# B&R Automation Studio project TD52 (part 23)

### module_AGPara.typ
```iecst
TYPE
	PARA_AG_struct : 	STRUCT
		tiFreshOilPump_Delay : TIME := T#5s; (*PARA [15065]  OilFill V4.14*) (*OldName: NewPV V4.14*)
		iOilRefill_Type : INT; (*PARA [xxxxx]  OilFill V4.14 prepared*) (*OldName: NewPV V4.14*)
		tiPostLub_Continuous : TIME; (*PARA [14930]  Turbocharger post lubrication - Duration of the continuous phase [s]*) (*OldName: new PV; Cycle:5*) (*V04.12.00.00*)
		iNum_PostLub_Interval : INT; (*PARA [14931]  Turbocharger post lubrication - number of intervals*) (*OldName: new PV; Cycle:5*) (*V04.12.00.00*)
		tiPostLub_PumpOff : TIME; (*PARA [14932]  Turbocharger post lubrication - Duration oil pump OFF [s]*) (*OldName: new PV; Cycle:5*) (*V04.12.00.00*)
		tiPostLub_PumpOn : TIME; (*PARA [14933]  Turbocharger post lubrication - Duration oil pump ON [s]*) (*OldName: new PV; Cycle:5*) (*V04.12.00.00*)
		bOilTankMonitoring : BOOL; (*PARA [14893]  OilTank V4.12*) (*OldName: NewPV V4.12*)
		rFreshOilTank_Type : REAL; (*PARA [14867]  OilTank V4.12*) (*OldName: NewPV V4.12*)
		rFreshOilTank_Length : REAL; (*PARA [14868]  OilTank V4.12*) (*OldName: NewPV V4.12*)
		rFreshOilTank_Height : REAL; (*PARA [14869]  OilTank V4.12*) (*OldName: NewPV V4.12*)
		rFreshOilTank_Witdh : REAL; (*PARA [14870]  OilTank V4.12*) (*OldName: NewPV V4.12*)
		rFreshOilTank_SensorPos : REAL; (*PARA [14871]  OilTank V4.12*) (*OldName: NewPV V4.12*)
		rWasteOilTank_Type : REAL; (*PARA [14876]  OilTank V4.12*) (*OldName: NewPV V4.12*)
		rWasteOilTank_Length : REAL; (*PARA [14877]  OilTank V4.12*) (*OldName: NewPV V4.12*)
		rWasteOilTank_Height : REAL; (*PARA [14878]  OilTank V4.12*) (*OldName: NewPV V4.12*)
		rWasteOilTank_Witdh : REAL; (*PARA [14879]  OilTank V4.12*) (*OldName: NewPV V4.12*)
		rWasteOilTank_SensorPos : REAL; (*PARA [14880]  OilTank V4.12*) (*OldName: NewPV V4.12*)
		rFreshOilTank_VolumeTotal : REAL; (*PARA [14894]  OilTank V4.12*) (*OldName: NewPV V4.12*)
		rWasteOilTank_VolumeTotal : REAL; (*PARA [14898]  OilTank V4.12*) (*OldName: NewPV V4.12*)
		rDayOilTank_VolumeTotal : REAL; (*PARA [14899]  OilTank V4.12*) (*OldName: NewPV V4.12*)
		rDayOilTank_Type : REAL; (*PARA [14885]  OilTank V4.12*) (*OldName: NewPV V4.12*)
		rDayOilTank_Length : REAL; (*PARA [14886]  OilTank V4.12*) (*OldName: NewPV V4.12*)
		rDayOilTank_Height : REAL; (*PARA [14887]  OilTank V4.12*) (*OldName: NewPV V4.12*)
		rDayOilTank_Witdh : REAL; (*PARA [14888]  OilTank V4.12*) (*OldName: NewPV V4.12*)
		rDayOilTank_SensorPos : REAL; (*PARA [14889]  OilTank V4.12*) (*OldName: NewPV V4.12*)
		rV_FreshOilTank_LimHi : REAL; (*PARA [14875]  OilTank V4.12*) (*OldName: NewPV V4.12*)
		rV_FreshOilTank_LimLo : REAL; (*PARA [14874]  OilTank V4.12*) (*OldName: NewPV V4.12*)
		rV_DayOilTank_LimHi : REAL; (*PARA [14875]  OilTank V4.12*) (*OldName: NewPV V4.12*)
		rV_DayOilTank_LimLo : REAL; (*PARA [14874]  OilTank V4.12*) (*OldName: NewPV V4.12*)
		rV_WasteOilTank_LimHi : REAL; (*PARA [14883]  OilTank V4.12*) (*OldName: NewPV V4.12*)
		rFreshOilTank_ScalMin : REAL; (*PARA [14872] [HalIO takeover]  OilTank V24*) (*OldName: NewPV V4.12*)
		rFreshOilTank_ScalMax : REAL; (*PARA [14873] [HalIO takeover]  OilTank V24*) (*OldName: NewPV V4.12*)
		rWasteOilTank_ScalMin : REAL; (*PARA [14881] [HalIO takeover]  OilTank V24*) (*OldName: NewPV V4.12*)
		rWasteOilTank_ScalMax : REAL; (*PARA [14882] [HalIO takeover]  OilTank V24*) (*OldName: NewPV V4.12*)
		rDayOilTank_ScalMin : REAL; (*PARA [14890] [HalIO takeover]  OilTank V24*) (*OldName: NewPV V4.12*)
		rDayOilTank_ScalMax : REAL; (*PARA [14891] [HalIO takeover]  OilTank V24*) (*OldName: NewPV V4.12*)
		bER_VentColdCountryMode : BOOL; (*PARA [12246]: engine room ventilation cold country mode *) (*OldName:MRL_KL; Cycle:5*)
		bPurgecycle_Active : BOOL; (*PARA [12256]: purge cycle enable*) (*OldName:bPurgecycle; Cycle:5*)
		bVISA : BOOL; (*PARA [12259]: monitoring according VISA*) (*OldName:VISA; Cycle:5*)
		bTSTC_Exist : BOOL; (*PARA [10018]: Engine with TSTC *) (*OldName:b2StageTC; Cycle:5*)
		bEngTyp3_Prelub_Active : BOOL; (*PARA [10009]: prelubrication for engine typ 3 active *) (*OldName:BR3_VS_aktiv; Cycle:5*)
		bTC_PostLub_Active : BOOL; (*PARA [10015]: turbo charger post lubrication active *) (*OldName:new; Cycle:5*)
		bBS_Acc_Active : BOOL; (*PARA [12178]: accelerated black start active *) (*OldName:sel_black_start_15s; Cycle:5*)
		bSel_TwoN2Valves : BOOL; (*PARA [11313]: select exhaust gas scavenging with 2 nitrogen*) (* OldName:TwoN2Valves; Cycle:5*)
		bECWP_MechDriven : BOOL; (*PARA [10007]: engine cooling water pump mechanical driven*) (*OldName:sel_BR3_eMKWP; Cycle:5*)
		bTC_watercooled : BOOL; (*PARA [10016]: water cooled turbo charger *) (*OldName:ATL_H2O; Cycle:5*)
		iEng_Motortype : INT; (* Motor type of the engine *) (*OldName:iMotortyp; Cycle:5*)
		rN_ECWP_Set : REAL; (*PARA [10032]: speed engine cooling water pump setpoint *) (* OldName:GW_SP_MKWP; Cycle:5*)
		rN_EngStart_HyHi : REAL; (*PARA [11295]: speed engine start limit high hysteresis *) (*OldName:HY_DREHZ; Cycle:5*)
		rN_EngStart_HyHiHi : REAL; (*PARA [11507]: speed engine start limit high high hysteresis *) (*OldName:HY_HDREHZ; Cycle:5*)
		rN_EngStartMon_LimHi : REAL; (*PARA [12068]: speed engine start monitoring limit high*) (*OldName:GW_STRDRE; Cycle:5*) (*V04.13.00.00*)
		rN_EngStart_LimHi : REAL; (*PARA [11296]: speed engine start limit high *) (*OldName:GW_DREHZ; Cycle:5*)
		rN_EngStart_LimHiHi : REAL; (*PARA [11508]: speed engine start limit high high *) (*OldName:GW_HDREHZ; Cycle:5*)
		rPr_CC_LimHiHi : REAL; (*PARA [10060]: pressure crank case limit high high *) (*OldName:GW_p_CC_high; Cycle:5*)
		bPr_CC_MS_Exist : BOOL; (*PARA [10013]: pressure crank case measuring signal exist *) (*OldName:p_CC_a; Cycle:5*)
		rPr_Prel1EOP_LimHi : REAL; (*PARA [10076]: prelubrication pressure limit for 1 pump*) (*OldName:GW_VSD1; Cycle:5*)
		rPr_Prel1EOP_HyHi : REAL; (*PARA [10075]: prelubrication pressure limit for 1 pump hysteresis*) (*OldName:HY_VSD1; Cycle:5*)
		rPr_Prel2EOP_LimHi : REAL; (*PARA [10078]: prelubrication pressure limit for 2 pump*) (*OldName:GW_VSD2; Cycle:5*)
		rPr_Prel2EOP_HyHi : REAL; (*PARA [10077]: prelubrication pressure limit for 2 pump hysteresis*) (*OldName:HY_VSD2; Cycle:5*)
		rPr_TCOF_PrelubMin : REAL; (*PARA [10087]: TC - filter outlet prelubrication pressure minimum*) (*OldName:GW_ODTC_MI_PREL; Cycle:5*)
		rPr_TCOF_PrelubHyMin : REAL; (*PARA [10086]: filter outlet prelubrication pressure minimum hysteresis*) (*OldName:HY_ODTC_MI_PREL; Cycle:5*)
		rT_ECW_PreH_HyOFF : REAL; (*PARA [10088]: temperature engine cooling water preheating limit off hysteresis *) (*OldName:HY_VORW; Cycle:5*)
		rT_ECW_PreH_LimOFF : REAL; (*PARA [10089]: temperature engine cooling water preheating limit off *) (*OldName:GW_VORW; Cycle:5*)
		bCtr_CC : BOOL; (*PARA [12644]: visibility crank case pressure controller*) (*OldName:new; Cycle:5*)
		bCtr_ECW : BOOL; (*PARA [10005]: visibility engine cooling water controller*) (*OldName:new; Cycle:5*)
		tCtr_CC : _tGeACtrPara; (*Para controller actual speed*) (*OldName:new; Cycle:5*)
		tCtr_ECW : _tGeACtrPara; (*Para controller engine cooling water temperature*) (*OldName:new; Cycle:5*)
		bTCOP_Visible : BOOL; (*PARA [10017]: turbo charger oil pump visible*) (*OldName:bVisuTCPump; Cycle:5*)
		bEOP_AC_Visible : BOOL; (*PARA [10010]: engine oil pump prelube AC visible*) (*OldName:bVisuACPump; Cycle:5*)
		bEOP_DC_Visible : BOOL; (*PARA [10011]: engine oil pump DC visible*) (*OldName:bVisuDCPump; Cycle:5*)
		bECW_PreH_Visible : BOOL; (*PARA [10006]: engine cooling water preheating visible*) (*OldName:bPreHeat; Cycle:5*)
		bECWP_PreH_Visible : BOOL; (*PARA [10008]: engine cooling water preheating pump visible*) (*OldName:bPreHeatWatPump; Cycle:5*)
		b_EOF_DiffMonActive : BOOL; (*PARA [10002]: Oil pressure before oil filter active M.03-PI-002(NUP29)*) (*OldName:bOilFilterPressAct; Cycle:5*)
		rN_EOP_Lim1 : REAL; (*PARA [10033]: Engine Speed 1 for oil pressure monitoring*) (*OldName:DR_ODR_1; Cycle:5*)
		rPr_EOP_HyMin : REAL; (*PARA [10070]: Oil pressure mimimum hysteresis*) (*OldName:HY_ODRA; Cycle:5*)
		rPr_EOP_HyLim1 : REAL; (*PARA [10068]: Oil pressure limit 1 hysteresis*) (*OldName:HY_ODGW1; Cycle:5*)
		rPr_EOP_LimMax : REAL; (*PARA [10072]: Oil pressure maximum*) (*OldName:GW_ODR_MAX; Cycle:5*)
		rPr_EOP_HyMax : REAL; (*PARA [10069]: Oil pressure maximum hysteresis*) (*OldName:HY_ODR_MAX; Cycle:5*)
		rPr_EOP_LimSpeed2 : REAL; (*PARA [10074]: Limit oil pressure at engine speed 2*) (*OldName:GW_ODR_2; Cycle:5*)
		rN_EngNom : REAL; (*PARA [12128]: engine nominal speed*) (*OldName:n_nenn; Cycle:5*)
		rN_TCOF_Lim1 : REAL; (*PARA [10037]: TC - filter outlet pressure minimum speed scale value 1 for pressure monitoring*) (*OldName:DR_ODR_TC_1; Cycle:5*)
		rN_TCOF_Lim2 : REAL; (*PARA [10038]: TC - filter outlet pressure minimum speed scale value 2 for pressure monitoring*) (*OldName:DR_ODR_TC_2; Cycle:5*)
		rPr_TCOF_LimSpeed1 : REAL; (*PARA [10082]: TC - filter outlet pressure minimum oil limit value 1 for pressure monitoring*) (*OldName:GW_ODR_TC_1; Cycle:5*)
		rPr_TCOF_LimSpeed2 : REAL; (*PARA [10083]: TC - filter outlet pressure minimum oil limit value 2 for pressure monitoring*) (*OldName:GW_ODR_TC_2; Cycle:5*)
		rPr_TCOF_HyMin : REAL; (*PARA [10080]: TC - filter outlet pressure minimum hysteresis*) (*OldName:HY_ODTC_MI; Cycle:5*)
		rPr_TCOF_MinWarn : REAL; (*PARA [10085]: TC - filter outlet pressure minimum warning*) (*OldName:GW_ODTC_MI_W; Cycle:5*)
		rPr_TCOF_HyMinWarn : REAL; (*PARA [10081]: TC - filter outlet pressure minimum warning hysteresis*) (*OldName:HY_ODTC_MI_W; Cycle:5*)
		rPr_TCOF_Max : REAL; (*PARA [10084]: TC - filter outlet pressure maximum*) (*OldName:GW_ODTC_MA; Cycle:5*)
		rPr_TCOF_HyMax : REAL; (*PARA [10079]: TC - filter outlet pressure maximum hysteresis*) (*OldName:HY_ODTC_MA; Cycle:5*)
		rT_EO_PreheatMin : REAL; (*PARA [10093]: Limit start oil pre warning*) (*OldName:GW_OILVORW; Cycle:5*)
		rT_EO_PreheatHyMin : REAL; (*PARA [10092]: Limit start oil pre warning hysteresis*) (*OldName:HY_OILVORW; Cycle:5*)
		rT_EO_LimMin : REAL; (*PARA [10091]: Oil temperature minimum *) (*OldName:GW_OTMI; Cycle:5*)
		rT_EO_LimHyMin : REAL; (*PARA [10090]: Oil temperature minimum hysteresis*) (*OldName:HY_OTMI; Cycle:5*)
		b_TCEO_HE2Ena : BOOL; (*PARA [10004]: Activate picture for second oil heat exchanger*) (*OldName:bVisuOil2stage; Cycle:5*)
		rEOP_PreLube_Set : REAL; (*PARA [12673]: speed setpoint engine oil pump prelubrication (frequency converter)*) (*OldName:GW_SP_OILP_PREL; Cycle:5*)
		rEOP_PreHeat_Set : REAL; (*PARA [12674]: speed setpoint engine oil pump preheating (frequency converter)*) (*OldName:GW_SP_OILP_PREH; Cycle:5*)
		r_OV_LimOpen : REAL; (*PARA [10029]: Limit oil valve open*) (*OldName:GW_OELVA; Cycle:5*)
		r_OV_HyLimOpen : REAL; (*PARA [10027]: Limit oil valve open hysteresis*) (*OldName:HY_OELVA; Cycle:5*)
		r_OV_LimClose : REAL; (*PARA [10028]: Limit oil valve close*) (*OldName:GW_OELVZ; Cycle:5*)
		r_OV_HyLimClose : REAL; (*PARA [10026]: Limit oil valve close hysteresis*) (*OldName:HY_OELVZ; Cycle:5*)
		r_EO_LevelLimMax : REAL; (*PARA [10024]: Oil level maximum*) (*OldName:GW_OMAX; Cycle:5*)
		r_EO_W_LevelLimMax : REAL; (*PARA [14966]: Oil level maximum warning [%]*) (*OldName: newPV ; Cycle:5*) (*V04.13.00.00*)
		r_EO_W_LevelLimMin : REAL; (*PARA [13964]: Oil level minimum warning*) (*OldName: newPV ; Cycle:5*)
		r_EO_LevelHyLimMax : REAL; (*PARA [10022]: Oil level maximum hysteresis*) (*OldName:HY_OMAX; Cycle:5*)
		r_EO_LevelLimMin : REAL; (*PARA [10025]: Oil level minimum*) (*OldName:GW_OMIN; Cycle:5*)
		r_EO_LevelHyLimMin : REAL; (*PARA [10023]: Oil level minimum hysteresis*) (*OldName:HY_OMIN; Cycle:5*)
		rT_EOF_DiffMonRel : REAL; (*PARA [10094]: Oil filter differential pressure monitoring - Oil temperature for release [degC]*) (*OldName:ssOilFilterPOilTemp; Cycle:5*)
		rPr_EOP_LimSpeed1 : REAL; (*PARA [10073]: Limit oil pressure at engine speed 1*) (*OldName:GW_ODR_1; Cycle:5*)
		rPr_EOP_Lim1 : REAL; (*PARA [10071]: Oil pressure limit 1*) (*OldName:GW_ODGW1; Cycle:5*)
		rPr_LimHeatRel : REAL; (*PARA [12807]: Pressure limit for release heating*) (*OldName:GW_druck_heizfreigabe; Cycle:5*)
		rN_EOP_Lim2 : REAL; (*PARA [10034]: Engine Speed 2 for oil pressure monitoring*) (*OldName:DR_ODR_2; Cycle:5*)
		b_OilActive : BOOL; (*PARA [10003]: oil counter exist*) (*OldName:bExistOilCounter; Cycle:5*)
		iNum_OilPulse : INT; (*PARA [10020]: Impulse valency*) (*OldName:ssOilPulseValue; Cycle:5*)
		bCtr_EOVal_Active : BOOL; (*PARA [12615]: engine oil cooler valve controller Active*) (*OldName:new; Cycle:5*)
		rT_EOP_LimMax : REAL; (*PARA [10097]: Oil temperature maximum *) (*OldName:GW_OTMA; Cycle:5*)
		rT_EOP_HyMax : REAL; (*PARA [10095]: Oil temperature maximum hysteresis*) (*OldName:HY_OTMA; Cycle:5*)
		rT_EOP_HyRelLoad : REAL; (*PARA [10096]: Oil temperature release load, load enabling hysteresis*) (*OldName:HY_OT_LFG; Cycle:5*)
		rT_EOP_LimRelLoad : REAL; (*PARA [10098]: oil temperature release load*) (*OldName:GW_OT_LFG; Cycle:5*)
		tCtr_EOVal : _tGeACtrPara; (*Para: structure for engine oil controller*) (*OldName:new; Cycle:5*)
		rP_Red_T_Oil_Start : REAL; (*PARA [10049]: power reduction oil temp. start [°C]*) (*OldName:Pred_OT_start; Cycle:5*)
		rP_Red_T_Oil_Rate : REAL; (*PARA [10048]: power reduction oil temp.rate [%]*) (*OldName:Pred_OT_rate; Cycle:5*)
		rPr_EOF_DiffMonLimit1 : REAL; (*PARA [10065]: Oil filter differential pressure monitoring - Oil filter service life limit [bar]*) (*OldName:ssOilFilterLimit1; Cycle:5*)
		rPr_EOF_DiffMonLimit2 : REAL; (*PARA [10066]: Oil filter differential pressure monitoring - Oil filter to be replaced [bar]*) (*OldName:ssOilFilterLimit2; Cycle:5*)
		rPr_EOF_DiffMonLimit3 : REAL; (*PARA [10067]: Oil filter differential pressure monitoring - Shutdown [bar]*) (*OldName:ssOilFilterLimit3; Cycle:5*)
		i_OilRefillBlocked : DINT; (*PARA [10019]: Number of operating hours until next refill*) (*OldName:slBlockOilRefill_Bh; Cycle:5*)
		bEO_Level_Active : BOOL; (*PARA [12805]: Engine oil level measuring active*) (*OldName:ALM[2576].ENABLE; Cycle:5*)
		bPr_EOF_After_Active : BOOL; (*PARA [12722]: Oil pressure after oil filter active M.03-PI-057*) (*OldName:new PV; Cycle:5*)
		bGridCode_Active : BOOL; (*PARA [11055]: Gride Code active*) (*OldName:bGridCode; Cycle:5*)
		bPr_TCOaF_Active : BOOL; (*PARA [10014]: pressure oil turbo charger after filter signal active*) (*OldName:new; Cycle:5*)
		bCtr_EOVal_LT_Active : BOOL; (*PARA [12705]: engine oil cooler LT valve controller Active*) (*OldName:new; Cycle:5*)
		tCtr_EOVal_LT : _tGeACtrPara; (*Para: structure for engine oil controller*)
		bT_EOaPump_Active : BOOL; (*PARA [12723]: engine oil temperature after pump active*)
		bPr_Oil_LPTC_In_A : BOOL; (*PARA [12724]: oil pressure LP turbo charger A inlet measuring active*)
		bPr_Oil_LPTC_In_B : BOOL; (*PARA [12725]: oil pressure LP turbo charger B inlet measuring active*)
		bPr_f_BbFilt_Exist : BOOL; (*PARA [12566]: Druck vor Blow-by Filter aktiv, Pressure before Blow-by filter	*)
		rP_CC_MonActive_LimHi : REAL; (*PARA [10047]: -Visu only- Kurbelgehaeusedruckueberwachung aktiv, Crank Case Pressure check active [% Pnom]*) (*Oldname: GW_P_CCM, Cycle:5 *)
		rPr_CC_Lo : REAL; (*PARA [12560]: Kurbelgehaeusedruck Minimum - Warnung, Crank Case Pressure Minimum Warning [bar]*)
		rPr_CC_Hi : REAL; (*PARA [12561]: Crank case pressure high - warning [bar]*)
		rP_Red_CC : REAL; (*PARA [12564]: Power reduction by Crank case pressure [% Pnom]*)
		rPc_BbBlower_Hi : REAL; (*PARA [12565]: Operating point blow by blower maximum [%]*)
		bPr_a_BbFilt_Exist : BOOL; (*PARA [12571]: pressure after blow by filter exist*)
		rDPr_BbFilt_Pstart : REAL; (*PARA [12618]: Blow by filter difference pressure start point for monitoring [% Pnom]*)
		rDPr_BbFilt_Lo_P1 : REAL; (*PARA [12619]: Blow by filter difference pressure new filter - lower load point [bar]*)
		rDPr_BbFilt_Lo_P2 : REAL; (*PARA [12620]: Blow by filter difference pressure new filter - full load [bar]*)
		rDPr_BbFilt_Hi_P1 : REAL; (*PARA [12621]: Blow by filter difference pressure charged filter - lower load point [bar]*)
		rDPr_BbFilt_Hi_P2 : REAL; (*PARA [12622]: Blow by filter difference pressure charged filter - full load [bar]*)
		tiPr_CC_Hi : TIME; (*PARA [12562]: Crank case pressure high - time until warning [s]*)
		tiPr_CC_HiHi : TIME; (*PARA [12563]: Crank case pressure high - time until error [s]*)
		bT_EO_Pan_Active : BOOL; (*PARA [12747]: engine oil temperature oil pan active*)
		bPr_TCObF_Active : BOOL; (*PARA [12742]: turbocharger oil pressure before filter active*)
		bPr_AirStarter_Tank_Exist : BOOL; (*PARA [12648]: air starter tank pressure exist *)
		rPr_AirStarter_Tank_Lo : REAL; (*PARA [10055]: air starter tank pressure minimum [bar] *)
		bPr_AirStarter_Supply_Exist : BOOL; (*PARA [12651]: air starter supply pressure exist	*)
		rPr_AirStarter_Supply_LoLo : REAL; (*PARA [10053]: air starter supply pressure minimum - error [bar] *)
		rPr_AirStarter_Supply_HiHi : REAL; (*PARA [10052]: air starter supply pressure maximum - error [bar] *)
		bN_AirStarter_Exist : BOOL; (*PARA [12654]: air starter speed exist	*)
		tiAirStarter_OnTime : TIME; (*PARA [10119]: air starter ON Time / Engaging Time (Einspurzeit) [ms]*)
		tiTC_Postlub : TIME; (*PARA [12775]: turbo charger postlube duration for water cooled TC [ms]*)
		bManAuxCtr_Active : BOOL; (*PARA [12917]: Manual operating auxiliaries control is active*)
		tiManAuxCtr_Max : TIME; (*PARA [12916]: Maximum release time of manual operating auxiliaries control*)
		tiFreshOilPump_Intervall : TIME; (*PARA [xxxxx]: time for run time intervall fresh oil pump*) (*OldName: NewPV V4.14*)
		tiFreshOilPump_Pause : TIME; (*PARA [xxxxx]: time for stop intervall fresh oil pump*) (*OldName: NewPV V4.14  SEE ALSO -->PARA [13308]: time for run time overload fresh oil pump*)
		tiFreshOilPump_RTC_Time : TIME; (*PARA [13308]: time for run time overload fresh oil pump*)
		rP_Red_TransformerWarning_Rate : REAL; (*PARA [13270]: transformer power reduction setpoint*)
		bP_Red_TransformerWarning_Sel : BOOL; (*PARA [13269]: activation transformer power reduction*)
		bPr_f_BbFilt_A_Exist : BOOL; (*PARA [13265]: pressure before blow-by filter aktiv*)
		bPr_f_BbFilt_B_Exist : BOOL; (*PARA [13266]: pressure before blow-by filter aktiv*)
		bPr_a_BbFilt_A_Exist : BOOL; (*PARA [13267]: pressure after blow by filter exist*)
		bPr_a_BbFilt_B_Exist : BOOL; (*PARA [13268]: pressure after blow by filter exist*)
		bCDP_Active : BOOL; (*PARA [13182]: Kondensorpumpe active*)
		bPr_EOaP_Active : BOOL; (*PARA [13398]: engine oil pressure after pump active M.03-PI-007*)
		rPr_EOaP_LimHi : REAL; (*PARA [13399]: engine oil pressure after pump limit high M.03-PI-007*)
		rPr_EOaP_LimHiHi : REAL; (*PARA [13400]: engine oil pressure after pump limit high high M.03-PI-007*)
		bOilFiltUnit_Exist : BOOL; (*PARA [13470]: oil filter unit existing*)
		bPr_OFUbFilt_Active : BOOL; (*PARA [13471]: pressure oil filter unit before filter M.03-PI-011*)
		bPr_OFUaFilt_Active : BOOL; (*PARA [13474]: pressure oil filter unit after filter M.03-PI-012*)
		bServicePrelub : BOOL; (*PARA [13827]: prelube with both oil pumps - service button*)
		rPr_EObF_LimHi : REAL; (*PARA [13962]: Oil pressure filter inlet maximum warning [bar] M.03-PI-002(NUP29)*)
		rPr_EObF_LimHiHi : REAL; (*PARA [13963]: Oil pressure filter inlet maximum alarm [bar] M.03-PI-002(NUP29)*)
		bPr_OFUbCentrifuge_Active : BOOL; (*PARA [13631]: pressure oil filter unit before centrifuge M.03-PI-008*)
		rDPr_OFU_Filt_LimHi : REAL; (*PARA [13477]: difference pressure oil filter unit - limit high*)
		rPr_OFUbFilt_Hi : REAL; (*PARA [13630]: pressure oil filter unit before filter - limit high*)
		rPr_OFUbCentrifuge_Hi : REAL; (*PARA [13634]: pressure oil filter unit before centrifuge - limit high*)
		bPr_TCO_Active : BOOL; (*PARA [14114]: pressure oil before turbo charger [bar]*)
		tiFSPreL : TIME; (*PARA [14166]: permanent prelubrication minimum operating time for faststart release*)
		rPr_TCO_FSPreL_LimHi : REAL; (*PARA [14167]: pressure oil before turbo charger limit high - permanent prelubrication [bar]*)
		rPr_TCO_FSPreL_LimLo : REAL; (*PARA [14169]: pressure oil before turbo charger limit low - fast start [bar]*)
		rN_TCO_FS : REAL; (*PARA [14168]: speed point fast start [rpm]*)
		rT_EO_PreH_FS_Min : REAL; (*PARA [14170]: limit low start oil preheating warning/fast start [°C]*)
		rT_EO_PreH_FS_HyMin : REAL; (*PARA [14171]: Limit low start oil preheating warning hysteresis/fast start [°C]*)
		rPr_EO_PreH_LimLo : REAL; (*Para: engine oil pressure limit low preheating [bar]*)
		rPr_EO_FSPreL_LimLo : REAL; (*PARA [14165]: engine oil pressure limit low permanent prelubrication [bar]*)
		tiReEngage : TIME; (*PARA [14065]: delay reengagement air starter*)
		bFSPreL_Act : BOOL; (*PARA [14208]: permanent prelubrication active*)
		bBbOp_EOP : BOOL; (*PARA [14172]: blowby fan operation with engine oil pump*)
		bPreLub_Interval_Enable : BOOL; (*PARA [14066]: Interval pre lubrication enable *)
		tiPreLub_Interval : TIME; (*PARA [13965]: interval time pre lubrication *)
		rPr_PreLub_Interval_Lim : REAL; (*PARA [13966]: engine interval pre lubrication pressure limit *)
		rU_StarterBat_Lo : REAL; (*PARA [13989]: Starter battery voltage minimum (UL) while battery test*)
		rU_StarterBat_Hi : REAL; (*PARA [13990]: Starter battery voltage high*)
		bACP_Enable : BOOL; (*PARA [13984]: Enable Active Cooling *)
		rT_ACP_ECW_sp : REAL; (*PARA [13985]: Active cooling program setpoint temperature engine cooling water system *)
		rT_ACP_EO_sp : REAL; (*PARA [13986]: Active cooling program setpoint temperature engine cooling water system *)
		rT_ACP_AirER_sp : REAL; (*PARA [13987]: Active cooling program setpoint temperature engine room ventilation *)
		rT_EO_LimHiHi : REAL; (*PARA [14180]: Oil temperature high high//SWAT920/5*)
		bECW_PreH_Fast : BOOL; (*PARA [14349]: Fast ECW heat-up active*)
		rT_ECW_HydrPreH_LimLo : REAL; (*PARA [14350]: Delta hydraulic pre-heating warning [°C]*)
		iECW_PreH_Int_Visible : INT; (*PARA [11902]: Pre-heating type jacket water (formerly: Internal heating)*)
		bT_HW_Su_PreH_ECW_Active : BOOL; (*PARA [12912]: Heating water temperature supply hydraulic ECW preheating measuring active*)
		bRedHWP_Active : BOOL; (*PARA [14345]: Activate redundant pump control for heating water pump *)
		bRedCCWP_Active : BOOL; (*PARA [14347]: Activate redundant pump control for charge cooler water pump *)
		bRedCC2WP_Active : BOOL; (*PARA [14346]: Activate redundant pump control for charge cooler 2 water pump *)
		bRedEmCWP_Active : BOOL; (*PARA [14348]: Activate redundant pump control for emergency cooler water pump *)
		iCnt_TC_Inspection_Hi : DINT; (*PARA [14408]: Threshold for turbocharger inspection after number of failed post cooling cycles*)
		rPr_TC_EOF_After_Avg_Lo : REAL; (*PARA [14409]: Lower threshold average oil pressure for TC post cooling*)
		rPr_TC_Oil_CoolDownInterrupt_Lo : REAL; (*PARA [14410]: Lower threshold oil pressure for OCTC post cooling interruption*)
		bDPr_ECWP_Mon_Active : BOOL; (*PARA [14425]: Measurement cooling water difference pressure over ECW pump active*)
		rDPr_ECWP_LoLo : REAL; (*PARA [14428]: Difference pressure cooling water over ECW pump minimum*)
		tiAirST_Interrupt : TIME; (*PARA [14445]: Air starter start up time for interrupting blocked start valve*)
		bBbBlower_Off_Active : BOOL; (*PARA [14483]: Blow-by blower reduced operation mode*)
		rP_Norm_BbBlower_off : REAL; (*PARA [14484]: Engine power limit for blow by blower off [% Pnom]*)
		tiPr_CC_HiWarn : TIME; (*PARA [14485]: Crankcase pressure maximum  delay until warning [s]*)
		tiPreLube : TIME; (*PARA [14504]: Prelubrication duration (normal prelube, not permanent)*)
		bEO_Management_Active : BOOL; (*PARA [14496]: oil management function active*)
		bCW_Management_Active : BOOL; (*PARA [14497]: coolant management function active*)
		iEO_PreH_Int_Visible : INT; (*PARA [14503]: Pre-heating type engine oil (formerly: Internal heating)*)
		iBatMon_Mode : INT; (*PARA [14490]: Battery voltage monitoring mode*)
		rU_BufferBat_Lo : REAL; (*PARA [14491]: Buffer battery voltage minimum (UL) while battery test*)
		rU_BufferBat_Idle_Lo : REAL; (*PARA [14492]: Buffer battery voltage minimum idle voltage (U0)*)
		rU_StarterBat_Idle_Lo : REAL; (*PARA [14493]: Starter battery voltage minimum idle voltage (U0)*)
		rU_StarterBat_Crank_Lo : REAL; (*PARA [14494]: Starter battery voltage minimum starter cranking (UL)*)
		tiU_StarterBat_MeasDelay : TIME; (*PARA [14501]: Test begin starter battery voltage starter cranking (UL)*)
		tiU_StarterBat_MeasTime : TIME; (*PARA [14502]: Test duration starter battery voltage starter cranking (UL)*)
		rPr_OFUbCentrifuge_Lo : REAL; (*PARA [14734]: Oil pressure oil centrifuge inlet minimum warning [bar]*)
		iOQS_Config : UINT; (*PARA [14726]: Oil quality sensor configuration*)
		rOQS_OC_ScalFreshOil : REAL; (*PARA [14727]: Oil quality sensor: Oil condition value fresh oil (=100% oil quality) [%]*)
		rOQS_OC_ScalAgedOil : REAL; (*PARA [14728]: Oil quality sensor: Oil condition value aged oil (=0% oil quality) [%]*)
		rOilQual_OQS_OC_LimLo : REAL; (*PARA [14729]: Oil quality sensor: Limit oil quality warning [%]*)
		rOilQual_OQS_OC_LimLo1 : REAL; (*PARA [14731]: Oil quality sensor: Limit oil quality critical warning [%]*)
		rOilQualTendency_OQS_OC_LimHi : REAL; (*PARA [14730]: Oil quality sensor: Limit oil quality tendency warning [%/100oph]*)
		rOilQualTendency_OQS_OC_LimHi1 : REAL; (*PARA [14732]: Oil quality sensor: Limit oil quality tendency critical warning [%/100oph]*)
		iOilSamplingNomOh : DINT; (*PARA [14733]: Oil quality sensor: Regular oil sampling interval [oph]*)
		rT_OQS_LimLo : REAL; (*PARA [14921]: Oil quality sensor: Limit oil quality operating temperature [degC]*)
		rU_StarterMonTtT_LimHi : REAL; (*PARA [14927]: Starter monitoring: Tooth to tooth upper limit starter battery voltage [V]*)
		rN_StarterMonTtT_LimLo : REAL; (*PARA [14928]: Starter monitoring: Tooth to tooth lower limit engine speed [rpm]*)
		tiStarterMonDuration : TIME; (*PARA [14929]: Starter monitoring: Tooth to tooth detection duration [s]*)
		bOilRefill_MonAct : BOOL; (*PARA [14967]: Oil refill - Monitoring active*) (*OldName: newPV ; Cycle:5*) (*V04.13.00.00*)
		rVol_OilRefill_Pct_EO_Level : REAL; (*PARA [14968]: Oil refill - Refill volume per % oil level [l]*) (*OldName: newPV ; Cycle:5*) (*V04.13.00.00*)
		rPc_OilRefill_VolTolerance : REAL; (*PARA [14969]: Oil refill - Refill volume tolerance [%]*) (*OldName: newPV ; Cycle:5*) (*V04.13.00.00*)
		rU_StarterMon_LimLo : REAL; (*PARA [15015]: Starter function voltage level [V]*) (*OldName: newPV ; Cycle:5*) (*V04.13.00.00*)
		tiStarterFunDuration : TIME; (*PARA [15016]: Starter function detection time [s]*) (*OldName: newPV ; Cycle:5*) (*V04.13.00.00*)
		bEO_PreH_Active : BOOL; (*PARA [15019]: Oil preheating active*) (*OldName: newPV ; Cycle:5*) (*V04.13.00.00*)
		rT_EO_PreH_EngStart : REAL; (*PARA [15020]: Oil preheating - Target temperature for engine start [degC]*) (*OldName: newPV ; Cycle:5*) (*V04.13.00.00*)
		rVolFlow_Marg : REAL; (*PARA [15071]: Volume flow margin [%]*) (*V04.14.00.00*)
		rVolEff_CrkSpeed : REAL; (*PARA [15073]: Volumetric efficiency at cranking speed [-]*) (*V04.14.00.00*)
		iVol_MinAir_SysPurge : UDINT; (*PARA [15074]: Minimum air volume required for system purge [lt]*) (*V04.14.00.00*)
		rST_Heatup_Fact : REAL; (*PARA [15075]: Starter heatup factor [s/s]*) (*V04.14.00.00*)
		tiST_CooldownConst : TIME; (*PARA [15076]: Starter cool down time constant [s]*) (*V04.14.00.00*)
		tiST_MaxDur_OverheatPrev : TIME; (*PARA [15077]: Maximum starting duration overheat prevention [s]*) (*V04.14.00.00*)
		rST_ReqOpTiAftCooldown : REAL; (*PARA [15078]: Required starter operating time after cooldown [%]*) (*V04.14.00.00*)
		iVol_PremxInSys : UDINT; (*PARA [15079]: Premixed volume of the engine intake system [lt]*) (*V04.14.00.00*)
		iVol_TolUnbrtMxMax : UDINT; (*PARA [15080]: Maximum tolerable unburnt mixture volume [lt]*) (*V04.14.00.00*)
		bEGScav_Active : BOOL; (*PARA [11303]: exhaust gas scavenging active *) (*OldName:sel_EGScav;Cycle:5*) (*V04.14.00.00*)
		tiEO_Refill_TimeMax : TIME; (*PARA [15067]: oil refill time maximum *) (*V04.14.00.00*)
		bEGScav_ifAuxV_ok : BOOL; (*PARA [11304]: exhaust gas scavenging if auxiliaries voltage supply ok*) (*OldName:sel_EGScav_if_AuxV_ok;Cycle:5*)
	END_STRUCT;
END_TYPE
```

### module_AGPerm.typ
```iecst
(********************************************************************
 * COPYRIGHT -- INNIO Company
 ********************************************************************
 * Paket: AuxiliariesGeneral
 * Datei: module_AGPerm.typ
 * Autor: zengeres
 * Erstellt: 14. Oktober 2013
 ********************************************************************
 * Datentypen des Pakets AuxiliariesGeneral
 ********************************************************************)

TYPE
	tPerm_AG_typ : 	STRUCT
		tStartStat : ARRAY[0..200]OF tStartStat_typ;
		StatCnt : DINT;
		rAG_PermValue1 : REAL; (*spare permanent value - replace with new vars of same lenght, when needed*)
		rAG_PermValue2 : REAL; (*spare permanent value - replace with new vars of same lenght, when needed*)
		rAG_PermValue3 : REAL; (*spare permanent value - replace with new vars of same lenght, when needed*)
		rAG_PermValue4 : REAL; (*spare permanent value - replace with new vars of same lenght, when needed*)
		rAG_PermValue5 : REAL; (*spare permanent value - replace with new vars of same lenght, when needed*)
		rAG_PermValue6 : REAL; (*spare permanent value - replace with new vars of same lenght, when needed*)
		rAG_PermValue7 : REAL; (*spare permanent value - replace with new vars of same lenght, when needed*)
		rAG_PermValue8 : REAL; (*spare permanent value - replace with new vars of same lenght, when needed*)
		rAG_PermValue9 : REAL; (*spare permanent value - replace with new vars of same lenght, when needed*)
		rAG_PermValue10 : REAL; (*spare permanent value - replace with new vars of same lenght, when needed*)
	END_STRUCT;
	tStartStat_typ : 	STRUCT
		tiStartTime : RTCtime_typ;
		tiStarterON_Max : TIME;
		tiStarterOFF : TIME;
		tiStartScav : TIME;
		rN_EngStart : REAL;
		tiStartDuration : TIME;
		iStartID : DINT;
		bStartSuccess : BOOL;
	END_STRUCT;
END_TYPE
```

### module_AG.var
```iecst
VAR
	IN_AG : IN_AG_struct;
	OUT_AG : OUT_AG_struct;
	MM2VIS : MM2VIS_struct;
	VIS2MM : VIS2MM_struct;
	Para : PARA_AG_struct;
	ParaFactoryDefault : PARA_AG_struct;
	pm : PARA_AG_struct;
	tCtr_ECW_In : _tGeACtrIn; (*engine cooling water controller*)
	tCtr_ECW_Out : _tGeACtrOut; (*engine cooling water controller*)
	xCtr_ECW : GeACtr; (*engine cooling water controller*)
	xEngType : EngType;
	bEOVal_DemOpen : BOOL := FALSE; (*demand for oil refill valve V4.14 (without TOF)*)
	bStart : BOOL; (*engine start command from vis-button*)
	bStop : BOOL; (*engine stop command from vis-button*)
	bOMSS_Scav : BOOL; (*engine operation mode*)
	bOMSS_MAT : BOOL; (*engine operation mode*)
	bOMSS_Test : BOOL; (*engine operation mode*)
	bOMSS_Aut : BOOL; (*engine operation mode*)
	bOMSS_Man : BOOL; (*engine operation mode*)
	bOMSS_Off : BOOL; (*engine operation mode*)
	bNoMon4BlackStart : BOOL; (*no monitoring for engine blackstart*)
	bSafetyLoopEngOk : BOOL; (*saftey loop engine ok*)
	AN_VORW : BOOL; (* Vorwärmtemperatur *)
	bStartErr : BOOL; (*auto start failed *)
	AT26 : BOOL; (* Störung Hilfsbetriebe *)
	AT26_PB : BOOL; (* Prüfzeit Hilfsbetriebe *)
	bECW_CV_Open : BOOL; (* engine cooling water temperature control valve opened *)
	bGnlTrip : BOOL;
	bGnlTrip1 : BOOL;
	bGnlTrip2 : BOOL;
	bGnlTrip3 : BOOL;
	bGnlWarning : BOOL;
	bLampHornTest : BOOL; (*button start lamp test*)
	bT114 : BOOL;
	BTRB_30M : BOOL; (* Betrieb + 30min *)
	M_DREHZ : BOOL; (* Startdrehzahl *)
	M_DREHZ_5s : BOOL; (* Startdrehzahl + 5s*)
	M_HDREHZ : BOOL; (* Hochlaufdrehzahl *)
	M_HUPEAUS : BOOL; (* Hupe abschalten *)
	NKOP : BOOL; (* Nachkühlpumpe *)
	RESET : BOOL; (* RESET *)
	STP_STRT : BOOL; (* Zahn auf Zahn --> Starter raus *)
	T_H_STRT : BOOL; (* Handstart max. *)
	T_HUPEAUS : BOOL; (* Timer für Hupe *)
	T_ST_MKWP : BOOL; (* St. Motorkühlwasserpumpe *)
	T57 : BOOL; (* Störung Hilfsbetriebe *)
	bPreLube_EngStaRel : BOOL; (*prelube engine start release*)
	V_DREHZ : BOOL; (* Verlängerung Drehzahl *)
	xTOF_MKWP_op : TOF;
	ZM_STHBT : BOOL; (* ZM Störung Hilfsbetriebe *)
	ZM_STRT : BOOL; (* Zwischenmerker *)
	xTON_Pr_PreLub : TON; (*prelube oil pressure monitoring activation*)
	xRS_Pr_PreLub_Lo : RS; (*prelube oil pressure low monitoring delay*)
	bPr_PreLub_Lo : BOOL; (*prelube oil pressure low*)
	bTC_PostLub : BOOL; (*TC post lubrivation running*)
	AN_ODGW1 : BOOL; (* Öldruck Grenzwert 1 *)
	AN_ODR_MAX : BOOL; (* Öldruck maximum *)
	AN_ODRA : BOOL; (* Öldruck minimum *)
	AN_ODRW : BOOL; (* Öldruck minimum warnend *)
	bErrMsOilCounter : BOOL; (*ERROR measurement signal Oil counter*)
	BTRB_60s : BOOL; (*engine operation + 60s*)
	FG_ODRUW : BOOL; (* Freigabe Öldrucküberwachung *)
	kwh : REAL; (*Kilowatt hour *)
	ODR_NKUEHL : BOOL; (*Oilpressure for aftercoolingrun not achieved*)
	OilCounter : ARRAY[0..19] OF tOilCounter; (*circular buffer*)
	OilPress_a_ATL_min_A : BOOL; (*Öldruck nach Turboladerölfilter min abstellung*)
	OilPress_a_ATL_min_A_prel : BOOL; (*Öldruck nach Turboladerölfilter min abstellung vorschmierung*)
	rOC_Consum : REAL; (*oil consumption during the last measurement*)
	rOC_DeltaOpHour : REAL; (*operating hours during the last measurement*)
	rP_OC_Avg : REAL;
	rP_OC_Energy : REAL;
	rDPr_EOF : REAL; (*Oil filter differential pressure*)
	rVol_OC : REAL;
	slOilCounterImpulse : DINT; (*oil counter impulse*)
	slOilRefill_Bh : DINT; (*operating hour up to the time of last oil refill*)
	tCtr_EOVal_In : _tGeACtrIn; (*engine oil cooler valve controller In*)
	tCtr_EOVal_LT_In : _tGeACtrIn; (*engine oil cooler LT valve controller In*)
	tCtr_EOVal_Out : _tGeACtrOut; (*engine oil cooler valve controller Out*)
	tCtr_EOVal_LT_Out : _tGeACtrOut; (*engine oil cooler LT valve controller Out*)
	ucIndexOil : USINT; (*index for circular buffer Oil counter*)
	ucModeRegister1 : USINT := 14; (*Mode Register 1 for NC 150 Modul (00001110 binär) Ölzählereingang auf positive Zählrichtung setzen*)
	ucResetRegister1 : USINT := 128; (*reset oil counter *)
	UW_ODR_MAX : BOOL; (* UW Öldruck maximum *)
	xCtr_EOVal : GeACtr; (*engine oil cooler valve controller, function block GeACtr *)
	xCtr_EOVal_LT : GeACtr; (*engine oil cooler LT valve controller, function block GeACtr *)
	Z_ODR : BOOL; (* Zuschalt. Öldruck-UW *)
	rAvgActiveEnergy : REAL; (*active energy average*)
	rAvgOilVolume : REAL; (*oil volume average*)
	rAvgVolumeEnergy : REAL; (*oil volume / active energy average*)
	bPr_OTC_Prelub : BOOL; (* TC prelube oil pressure - release engine start*)
	b_OilRefillBlocked : BOOL; (* Blocking oil refill for X operating hours *) (*OldName:bBlockOil_Bh, Cycle:5*)
	bEO_Level_Hi : BOOL; (*engine oil level high from analog signal *) (*OldName:OMAX_fill; Cycle:5;*)
	bEO_Level_W_Hi : BOOL; (*engine oil level high from analog signal - warning*)
	bEO_Level_Lo : BOOL; (*engine oil level low from analog signal *) (*OldName:OMIN_fill; Cycle:5;*)
	bEO_Refill : BOOL; (*Oil refill valve open, builded from analog level sensor*) (*OldName:OELV_fill; Cycle:5;*)
	bPreHeatDem : BOOL; (*engine preheating demand*)
	bPreLubeDem : BOOL; (* engine prelubrication demand *) (*OldName:M_VORS, Cycle:5*)
	bTC_CoolDownRun : BOOL; (* turbo charger cool down run *) (*OldName:M_NKUEHL, Cycle:5*)
	bNoInitDetected : BOOL; (*allways true, except 1cycle on init up*)
	bTestEnabled : BOOL; (*Modultest enabled*)
	VORW_OIL : BOOL; (*engine oil preheating*) (*OldName:VORW_OIL, Cycle:5*)
	Perm : tPerm_AG_typ;
	bAMM_Pr_CC_MsMs : BOOL; (*W3323 Crank case pressure measuring signal failure*)
	bAMM_Pr_CC_Lo : BOOL; (*W2649 Crank case pressure low*)
	bAMM_Pr_CC_Hi : BOOL; (*W2558 Crank case pressure high*)
	bAMM_Pr_CC_HiHi : BOOL; (*W3322 Crank case pressure high*)
	bAMM_Pc_BbBlower_Hi : BOOL; (*W2591 Blow by blower speed maximum*)
	bAMM_BbBlower_Not_Rdy : BOOL; (*W2650 Blow by blower not ready*)
	bAMM_Pr_f_BbFilt_Ms : BOOL; (*W2651 Measuring signal failure pressure before blow by filter*)
	bAMM_Pr_f_BbFilt_A_Ms : BOOL; (*W2754 Measuring signal failure pressure before blow by filter A*)
	bAMM_Pr_f_BbFilt_B_Ms : BOOL; (*W2755 Measuring signal failure pressure before blow by filter B*)
	bAMM_Pr_a_BbFilt_Ms : BOOL; (*W2652 Measuring signal failure pressure after blow by filter*)
	bAMM_Pr_a_BbFilt_A_Ms : BOOL; (*W2756 Measuring signal failure pressure after blow by filter A*)
	bAMM_Pr_a_BbFilt_B_Ms : BOOL; (*W2757 Measuring signal failure pressure after blow by filter B*)
	bAMM_DPr_BbFilt_Hi : BOOL; (*W2653 Blow by filter difference pressure high - maintenance*)
	bAMM_DPr_BbFilt_A_Hi : BOOL; (*W2758 Blow by filter difference pressure high A - maintenance*)
	bAMM_DPr_BbFilt_B_Hi : BOOL; (*W2759 Blow by filter difference pressure high B - maintenance*)
	bAMM_DPr_BbFilt_Lo : BOOL; (*W2654 Blow by filter difference pressure low*)
	bAMM_DPr_BbFilt_A_Lo : BOOL; (*W2760 Blow by filter difference pressure low A*)
	bAMM_DPr_BbFilt_B_Lo : BOOL; (*W2761 Blow by filter difference pressure low B*)
	bAMM_MaxDC_Time : BOOL; (*W2427 Maximum allowed prelub time with DC pump exeeded*)
	rDPr_BbFilt : REAL := 0.0; (*calculated blow-by filter difference pressure*)
	rDPr_BbFilt_A : REAL := 0.0; (*calculated blow-by filter difference pressure bank A*)
	rDPr_BbFilt_B : REAL := 0.0; (*calculated blow-by filter difference pressure bank B*)
	tCtr_CC_In : _tGeACtrIn; (*Actual Speed BlowBy*)
	tCtr_CC_Out : _tGeACtrOut; (*Actual Speed BlowBy*)
	xCtr_CC : GeACtr; (*Actual Speed BlowBy*)
	rPc_BbBlower : REAL := 0.0; (*actual operating point blow by blower [%]*)
	bAMM_Pr_bEOF_Ms : BOOL; (*Measuring signal failure oil pressure before oil filter*)
	bAMM_Pr_aEOF_Ms : BOOL; (*Measuring signal failure oil pressure after oil filter*)
	bAMM_Pr_EngLubOil_Ms : BOOL; (*Measuring signal failure oil pressure engine lube oil*)
	bAMM_DPr_EOF_Lim1 : BOOL; (*Oil filter differential pressure - Oil filter achieves service life limit*)
	bAMM_DPr_EOF_Lim2 : BOOL; (*Oil filter differential pressure - Oil filter to be replaced*)
	bAMM_DPr_EOF_Lim3 : BOOL; (*Oil filter differential pressure - Maximum*)
	bAMM_Pr_AirStarter_Tank_Ms : BOOL; (* measuring signal failure air starter tank pressure - warning	*)
	bAMM_Pr_AirStarter_Tank_Lo : BOOL; (* air starter tank pressure minimum - warning		*)
	bAMM_Pr_AirStarter_Tank_LoLo : BOOL; (* air starter tank pressure minimum - error		*)
	bAMM_Pr_AirStarter_Supply_MsMs : BOOL; (* measuring signal failure air starter supply pressure - error	*)
	bAMM_Pr_AirStarter_Supply_LoLo : BOOL; (* air starter supply pressure minimum - error	*)
	bAMM_Pr_AirStarter_Supply_HiHi : BOOL; (*	air starter supply pressure maximum - error	*)
	bAMM_Pr_AirST_Engage_Ms : BOOL; (*Measurement signal failure pressure air starter engagement*)
	bAMM_AirStarter_StartUp : BOOL; (* air starter start up failure - error	*)
	rN_AirStarter : REAL; (* Air starter speed [rpm]*)
	bMsg1292_Set : BOOL; (*Manual operating auxiliaries control (Handbedienebene) active *)
	bECW_PreHV_Active : BOOL;
	bAMM_DPr_OFU_Filt_Hi : BOOL := FALSE; (*oilfilter difference pressure (oil filter unit) high - warning*)
	bPr_EO_PcheckFail : BOOL; (*plausibility check measuring signal //SWAT920/5*)
	iCntH : DINT; (*service mode operating hours*)
	iCntS : DINT; (*service mode starts*)
	bServicePrelube : BOOL; (*service mode prelubrication*)
	bAMM_DPr_OFU_Filt_HiHi : BOOL := FALSE; (*oilfilter difference pressure (oil filter unit) high + 2 bar*)
	bAMM_Pr_OFUbFilt_Hi : BOOL := FALSE; (*oil pressure before filter (oil filter unit) maximum - warning*)
	bAMM_Pr_OFUbCentrifuge_Hi : BOOL := FALSE; (*oil pressure before centrifuge (oil filter unit) maximum - warning*)
	bPreLubeDemFS : BOOL; (*permanent prelubrication demanded for fast start*)
	bAMM_EngageErr : BOOL; (*air starter engage error - fast start*)
	bEO_Level_W_Lo : BOOL; (* SWAT#3 *)
	AN_OD_AF_RA : BOOL; (* SWAT#3 *)
	AN_VSD1 : BOOL := 0; (*prelube pressure limit 1 pump*)
	AN_VSD2 : BOOL := 0; (*prelube pressure limit 2 pumps*)
	xTOF_ShortPreLubeTime_Delay : TOF; (* engine short pre lubrication with off cycle delay *)
	xTON_StarterBat_Hi : TON; (* starter battery voltage maximum timer *)
	tRealTime : rtctime_typ;
	bACP_Start : BOOL; (* Active Cooling Program start *)
	bACP_Cmp : BOOL; (* Active Cooling Program completed *)
	bACP_ECW_Cmp : BOOL; (* Active Cooling Program Engine Cooling Water completed *)
	bACP_EO_Cmp : BOOL; (* Active Cooling Program Engine Oil completed *)
	bPr_EOaF_PcheckFail : BOOL; (*plausibility check measuring signal//SWAT920/5a*)
	bEmLubDem : BOOL; (*emergency lubrication demanded*)
	bOCTC_CoDoRun : BOOL; (*oil cooled TC cool down run*)
	bWCTC_CoDoRun : BOOL; (*water cooled TC cool down run*)
	xTOF_OCTC_CoolDown : TOF; (*TOF oil cooled TC cool down run*)
	xTOF_WCTC_CoolDown : TOF; (*TOF water cooled TC cool down run*)
	xTOF_WCTC_PostLub : TOF; (*TOF water cooled TC post*)
	iCnt_TL : INT := 0; (*J920: TC interval cooldown program pulse number *)
	xTON_TL_OP_Aus : TON := (0); (*J920: TC interval cooldown program off pulse*)
	xTON_TL_OP_Ein : TON := (0); (*J920: TC interval cooldown program on pulse*)
	xTP_StartFail : TP; (*delay messages in case of a failed start attempt*)
	rT_ECW_HydrPreH_LimLo : REAL; (*Temperature limit ECW heat-up/hydraulic pre-heating failure warning*)
	xSR_PreH_HeatUpDone : SR;
	bECW_HydrPreH_Dem : BOOL; (*ECW hydraulic pre-heating demand*)
	bRedHWP_Fail : BOOL; (*Redundant heating water pump failure*)
	bRedCCWP_Fail : BOOL; (*Redundant water pump failure charge cooler*)
	bRedCC2WP_Fail : BOOL; (*Redundant water pump failure charge cooler 2*)
	bRedEmCWP_Fail : BOOL; (*Redundant water pump failure emergency cooling circuit*)
	iRedHWP_Fail : INT; (*Redundant heating water pump fault indication/pump ID*)
	iRedCCWP_Fail : INT; (*Redundant charge cooler water pump fault indication/pump ID*)
	iRedCC2WP_Fail : INT; (*Redundant charge cooler 2 water pump fault indication/pump ID*)
	iRedEmCWP_Fail : INT; (*Redundant emergency cooler water pump fault indication/pump ID*)
	bAMM_Pr_AirST_Engage_Lo : BOOL; (*pressure air starter engagement minimum - error		*)
	iCnt_TC_abs : DINT; (*absolute counter for failed post cooling of the turbocharger*)
	iCnt_TC_rel_A : DINT; (*relative counter for failed post cooling of the turbocharger on bank A*)
	iCnt_TC_rel_B : DINT; (*relative counter for failed post cooling of the turbocharger on bank B*)
	iSt_TC_PwrInterrupt : DINT; (*permanent variable for TC black sut-down interruption by PLC power supply failure*)
	iCnt_TC_abs_RSP : DINT; (*absolute counter for failed post cooling of the turbocharger caused by DIANE power interruption*)
	bTC_CoolDownInterrupt : BOOL; (* TC post-cooling interruption *)
	xTON_RM_VWP : TON; (*TON feedback signal of flow switch in ECW circuit for pre-heating*)
	T_RM_VWP : BOOL; (*water flow in ECW circuit sufficient for pre-heating*)
	bECWP_Op_DPr_Mon : BOOL; (*ECWP operation status for pump monitoring via difference pressure*)
	tPr_TCLubOil_Min : HALioAi_Type; (*selection of TC lubrication oil pressure sensor for minimum monitorings*)
	tPr_TCLubOil_Max : HALioAi_Type; (*selection of TC lubrication oil pressure sensor for maximum monitorings*)
	xTON_ECWP_MonFS : TON; (*delayed operation monitoring of ECWP for fast start*)
	bPr_TCLubOil_PreL_FS_Hi : BOOL; (*W9221/W9224 turbocharger oil pressure high - permanent prelubrication*)
	bPr_TCLubOil_PreL_FS_HiHi : BOOL; (*W9222/W9225 turbocharger oil pressure high - permanent prelubrication OFF*)
	bMsg9002_set : BOOL;
	bMsg9001_set : BOOL;
	bMsg9332_set : BOOL;
	bMsg9048_set : BOOL;
	bMsg9003_set : BOOL;
	bMsg9333_set : BOOL;
	bStarterBat_Disconnect : BOOL;
	bChargeOff_EngStart : BOOL;
	bAMM_U_StarterBat_Lo : BOOL;
	bAMM_U_BufferBat1_Lo : BOOL;
	bAMM_U_BufferBat2_Lo : BOOL;
	iNr_CtrlBat_Used : USINT;
	bAMM_U_CtrlBat_Lo_Coll : BOOL;
	bAMM_Pr_OFUbCentrifuge_Lo : BOOL;
	bStartScavBgnFroce : BOOL; (*scavenging forced at the beginning of start attempt*)
	bStartScavFail : BOOL; (*Scavenging by starter motor failure*)
	bStartScavBgn : BOOL; (*Scavenging procedure anticipated at the beginning of the start attempt*)
	bStartScavUnsfl : BOOL; (*Scavenging by starting system not succesful*)
	bStartScavSflMsg : BOOL; (*Scavenging by starting system successful*)
	iVol_PurgeAir : UDINT; (*volume of purge air [lt]*)
	bSt_Purge : BOOL; (*purge state (true: engine purged, false: engine not purged)*)
	bSfl_PurgeCrk : BOOL; (*purge cranking cycle successful*)
	bFail_PurgeCrk : BOOL; (*purge cranking cycle unsuccessful*)
	bFail_StartAtt : BOOL; (*start attempt uncussessful*)
	bPreLubeOff_STT : BOOL; (*stop prelubrication due to start overheat*)
	bMsg9096_enable : BOOL; (*B9096 starter overheated enable*)
	bMsg9096_set : BOOL; (*B9096 starter overheated set*)
	bMsg9096_iTi_ST_UntRelDur : DINT; (*B9096 starter overheated duration until release [s]*)
	bMsg9097_set : BOOL; (*B9097 purge cranking cycle initiated set*)
	bMsg2376_T6_set : BOOL; (*A2376 purge cranking cycle T6 unsuccessful*)
	bMsg2382_set : BOOL; (*A2382 start attempt failed minimum speed*)
	bMsg9088_T6_set : BOOL; (*B9088 purge cranking cycle T6 successful*)
	xR_TRIG_bEng_Dem_Aut : R_TRIG; (*demand automatic mode rising egde*)
	iTi_ST_Res : INT; (*remaining starting time [s]*)
	bStartErr_ST_UntRelDur_High : BOOL; (*Start up failure due to starter overheat*)
	xTP_bMsg9096_set_retain : TP; (*message 9096 retain in case of start up failure*)
	bAMM_OQS_OC_ValueLo : BOOL;
	bAMM_OQS_OC_ValueLo1 : BOOL;
	bAMM_OQS_OC_TendencyHi : BOOL;
	bAMM_OQS_OC_TendencyHi1 : BOOL;
	bAMM_OQS_OC_MSF : BOOL;
	bOpMsg_ExtendOilSampleOh : BOOL;
	bAMM_Vol_OilRefill_Hi : BOOL := FALSE; (*W9378 Oil refill volume maximum *)
	bAMM_T_EO_PreH_EngStart_Lo : BOOL := FALSE; (*W9390 Oil temperature before engine start too low*)
	bAMM_9513 : BOOL; (*W9513 Failure engine oil refilling*)
END_VAR
VAR CONSTANT
	iNum_CtrlBatMon : USINT := 4; (*number of control battery monitoring test sets*)
END_VAR
VAR
	bCtrlBat_Used : ARRAY[1..iNum_CtrlBatMon] OF BOOL; (*Control battery set [x] used*)
END_VAR
VAR CONSTANT
	iOQS_OC_OilCfg_ByteSize : UINT := 380; (*number of byte of OilCfg string (2 hex char = 1 byte)*)
	iOQS_OC_OilCfg_CharSize : UINT := 2*iOQS_OC_OilCfg_ByteSize; (*number of hex char of OilCfg string (2 hex char = 1 byte)*)
	iOQS_OC_OilSerialNr_ByteSize : UINT := 14; (*number of byte of OilSerialNr string (2 hex char = 1 byte)*)
	iOQS_OC_OilSerialNr_CharSize : UINT := 2*iOQS_OC_OilSerialNr_ByteSize; (*number of hex char of OilSerialNr string (2 hex char = 1 byte)*)
END_VAR
VAR
	bEleStarterFail_Num : ARRAY[0..3] OF BOOL; (*starters failure array*)
END_VAR
```

### Program Logical/AuxiliariesGeneral/default_AG (IEC, version 4.14.0) - default

#### default_AGCyclic.st
```iecst
(*******************************************************************************
default		value set

This code is confidential and proprietary to the INNIO Company.
It may not be used in any form, or reproduced in any manner,
without the express written permission of the INNIO Company.
Copyright, INNIO Company, 2025

Customized modifications: -
------------------------

History:
-------
V4.00.0	24.04.2012	lettenb.	new
		01.10.2014  			tEO_Level_Hi/Lo removed(setted for 2times)
V4.00.1	29.01.2015  			920(stapelfeld) added
V4.03.0 29.07.2015	plattner	DayOil.. added
		13.10.2015	lettenb.	oiltank.. added
V4.04.0 09.05.2016				tCV_..., tL_OilSump3Hi added
		07.09.2016	Tinello		oil filter unit added
V4.06.0	19.06.2018	Perktold,	Louvers closed messages
V4.07.0 09.08.2018	Schmid		tCC2WP_Op added
		08.01.2019	Schmid		redundant pump control
		10.01.2019	Schmid		boiler failure and seismic alarm added
		25.02.2019	Stary/lett. bAuxRel_FireProtFlaps: FireProtFlap feedback signals included in aux.release, safety case
V4.10.0 26.05.2020	Schmid		tECWP_CB_On added
		24.11.2020	lettenb.	grid config.monitoring added
		18.01.2021	Schmid		sensors for leakage detection in additional external oil tank
V4.11.0 17.12.2021	Schmid		control battery check
		17.01.2022	lettenb.	tInAirER_Lou1/2, tOutAirER_Lou removed, bugfix
V4.14.0 11.04.2025	Tinello		SAFETY related:	tSafetyLoop_EmStop and tSafetyLoop_Eng added to get rid of problems during simulation

Instructions for use:
--------------------
Outstandings:
------------
*******************************************************************************)
PROGRAM _CYCLIC

	(* default TRUE setting for not existing Di's *)
	IN_AG.tSafetyLoop_EmStop.Di		:=	IN_AG.tSafetyLoop_EmStop.Di		OR  NOT IN_AG.tSafetyLoop_EmStop.GoodQual; 	(* SAFETY PLC *)
	IN_AG.tSafetyLoop_Eng.Di		:=	IN_AG.tSafetyLoop_Eng.Di		OR  NOT IN_AG.tSafetyLoop_Eng.GoodQual; 	(* SAFETY PLC *)
	IN_AG.tL_ECW_Lo.Di				:=	IN_AG.tL_ECW_Lo.Di				OR	NOT IN_AG.tL_ECW_Lo.GoodQual;
	IN_AG.tL_ECW_LoLo.Di			:=	IN_AG.tL_ECW_LoLo.Di			OR	NOT IN_AG.tL_ECW_LoLo.GoodQual;
	IN_AG.tCP_CBTrip.Di				:=	IN_AG.tCP_CBTrip.Di				OR	NOT IN_AG.tCP_CBTrip.GoodQual;
	IN_AG.tIFCP_CBTrip.Di			:=	IN_AG.tIFCP_CBTrip.Di			OR	NOT IN_AG.tIFCP_CBTrip.GoodQual;
	IN_AG.tMCP_CBTrip.Di			:=	IN_AG.tMCP_CBTrip.Di			OR	NOT IN_AG.tMCP_CBTrip.GoodQual;
	IN_AG.tU_StarterBat_Lo.Di		:=	IN_AG.tU_StarterBat_Lo.Di		OR	NOT IN_AG.tU_StarterBat_Lo.GoodQual;
	IN_AG.tL_WasteOilTank_Hi.Di		:=	IN_AG.tL_WasteOilTank_Hi.Di		OR	NOT IN_AG.tL_WasteOilTank_Hi.GoodQual;
	IN_AG.tAuxOverVoltProt_Ok.Di	:=	IN_AG.tAuxOverVoltProt_Ok.Di	OR	NOT IN_AG.tAuxOverVoltProt_Ok.GoodQual;
	IN_AG.tUPS_Ok.Di				:=	IN_AG.tUPS_Ok.Di				OR	NOT IN_AG.tUPS_Ok.GoodQual;
	IN_AG.tT_AirIFCP_Hi.Di			:=	IN_AG.tT_AirIFCP_Hi.Di			OR	NOT IN_AG.tT_AirIFCP_Hi.GoodQual;

	IN_AG.tAuxV_Eng_ok.Di			:=	IN_AG.tAuxV_Eng_ok.Di			OR	NOT IN_AG.tAuxV_Eng_ok.GoodQual;
	IN_AG.tEOP1AC_CB_trip.Di		:=	IN_AG.tEOP1AC_CB_trip.Di		OR	NOT IN_AG.tEOP1AC_CB_trip.GoodQual;
	IN_AG.tFS_ECW.Di				:=	IN_AG.tFS_ECW.Di				OR	NOT IN_AG.tFS_ECW.GoodQual;
	IN_AG.tGT1_SafeDevOK.Di			:=	IN_AG.tGT1_SafeDevOK.Di			OR	NOT IN_AG.tGT1_SafeDevOK.GoodQual;
	IN_AG.tGT2_SafeDevOK.Di			:=	IN_AG.tGT2_SafeDevOK.Di			OR	NOT IN_AG.tGT2_SafeDevOK.GoodQual;
	IN_AG.tRelAuxNoMon.Di			:=	IN_AG.tRelAuxNoMon.Di			OR	NOT IN_AG.tRelAuxNoMon.GoodQual;
	IN_AG.tMainsStartDevOk.Di		:=	IN_AG.tMainsStartDevOk.Di		OR	NOT IN_AG.tMainsStartDevOk.GoodQual;
	IN_AG.tEO_Level_Hi.Di			:=	IN_AG.tEO_Level_Hi.Di			OR	NOT IN_AG.tEO_Level_Hi.GoodQual;
	IN_AG.tEO_Level_Lo.Di			:=	IN_AG.tEO_Level_Lo.Di			OR	NOT IN_AG.tEO_Level_Lo.GoodQual;
	IN_AG.tCDP_Op.Di				:=	IN_AG.tCDP_Op.Di				OR	NOT IN_AG.tCDP_Op.GoodQual;
	IN_AG.tEOP_Op.Di				:=	IN_AG.tEOP_Op.Di				OR	NOT IN_AG.tEOP_Op.GoodQual;
	IN_AG.tGasAlarm.Di				:=	IN_AG.tGasAlarm.Di				OR	NOT IN_AG.tGasAlarm.GoodQual;
	IN_AG.tGasPreAlarm.Di			:=	IN_AG.tGasPreAlarm.Di			OR	NOT IN_AG.tGasPreAlarm.GoodQual;
	IN_AG.tFireAlarm.Di				:=	IN_AG.tFireAlarm.Di				OR	NOT IN_AG.tFireAlarm.GoodQual;
	IN_AG.tRelMainGVext.Di			:=	IN_AG.tRelMainGVext.Di			OR	NOT IN_AG.tRelMainGVext.GoodQual;
	IN_AG.tMainsStartDevFail.Di		:=	IN_AG.tMainsStartDevFail.Di		OR	NOT IN_AG.tMainsStartDevFail.GoodQual;
	IN_AG.tU_StarterBat_Lo.Di		:=	IN_AG.tU_StarterBat_Lo.Di		OR	NOT IN_AG.tU_StarterBat_Lo.GoodQual;
	IN_AG.tECWP_FC_Rdy.Di			:=	IN_AG.tECWP_FC_Rdy.Di			OR	NOT IN_AG.tECWP_FC_Rdy.GoodQual;
	IN_AG.tEOP_FC_Rdy.Di			:=	IN_AG.tEOP_FC_Rdy.Di			OR	NOT IN_AG.tEOP_FC_Rdy.GoodQual;
	IN_AG.tAuxFail.Di				:=	IN_AG.tAuxFail.Di				OR	NOT IN_AG.tAuxFail.GoodQual;
	IN_AG.tTransformerTrip.Di		:=	IN_AG.tTransformerTrip.Di		OR	NOT IN_AG.tTransformerTrip.GoodQual;
	IN_AG.tTransformerWarning.Di	:=	IN_AG.tTransformerWarning.Di	OR	NOT IN_AG.tTransformerWarning.GoodQual;
	IN_AG.tSafetyLoop_Gas.Di		:=	IN_AG.tSafetyLoop_Gas.Di		OR	NOT IN_AG.tSafetyLoop_Gas.GoodQual;
	IN_AG.tSafetyLoop_HWC.Di		:=	IN_AG.tSafetyLoop_HWC.Di		OR	NOT IN_AG.tSafetyLoop_HWC.GoodQual;
	IN_AG.tL_OilSumpHi.Di			:=	IN_AG.tL_OilSumpHi.Di			OR	NOT IN_AG.tL_OilSumpHi.GoodQual;
	IN_AG.tL_OilSump2Hi.Di			:=	IN_AG.tL_OilSump2Hi.Di			OR	NOT IN_AG.tL_OilSump2Hi.GoodQual;
	IN_AG.tL_OilSump3Hi.Di			:=	IN_AG.tL_OilSump3Hi.Di			OR	NOT IN_AG.tL_OilSump3Hi.GoodQual;

	IN_AG.tEOF_DiffMax.Di 			:= IN_AG.tEOF_DiffMax.Di 			OR NOT IN_AG.tEOF_DiffMax.GoodQual;
    IN_AG.tPr_TCOF_EOF_DiffMax.Di 	:= IN_AG.tPr_TCOF_EOF_DiffMax.Di 	OR NOT IN_AG.tPr_TCOF_EOF_DiffMax.GoodQual;
 	IN_AG.tPr_EO_Gear_Min.Di		:= IN_AG.tPr_EO_Gear_Min.Di 		OR NOT IN_AG.tPr_EO_Gear_Min.GoodQual;
	IN_AG.tT_EO_Gear_Max.Di			:= IN_AG.tT_EO_Gear_Max.Di			OR NOT IN_AG.tT_EO_Gear_Max.GoodQual;
	IN_AG.tEO_Supply_Fail.Di		:= IN_AG.tEO_Supply_Fail.Di			OR NOT IN_AG.tEO_Supply_Fail.GoodQual;

	IN_AG.tCO_Alarm.Di				:= IN_AG.tCO_Alarm.Di				OR NOT IN_AG.tCO_Alarm.GoodQual;
	IN_AG.tCO_PreAlarm.Di			:= IN_AG.tCO_PreAlarm.Di			OR NOT IN_AG.tCO_PreAlarm.GoodQual;
	IN_AG.tAuxErrWarn.Di			:= IN_AG.tAuxErrWarn.Di				OR NOT IN_AG.tAuxErrWarn.GoodQual;
	IN_AG.tActFiltAlarm.Di			:= IN_AG.tActFiltAlarm.Di			OR NOT IN_AG.tActFiltAlarm.GoodQual;
	IN_AG.tActFiltWarn.Di			:= IN_AG.tActFiltWarn.Di			OR NOT IN_AG.tActFiltWarn.GoodQual;
	IN_AG.tL_InMa_NotHi.Di			:= IN_AG.tL_InMa_NotHi.Di			OR NOT IN_AG.tL_InMa_NotHi.GoodQual;

	IN_AG.tECWP_Op.Di				:= IN_AG.tECWP_Op.Di				OR NOT IN_AG.tECWP_Op.GoodQual;
	IN_AG.tEngTurn.Di				:= IN_AG.tEngTurn.Di				OR NOT IN_AG.tEngTurn.GoodQual;
	IN_AG.tTCOP_CB_On.Di			:= IN_AG.tTCOP_CB_On.Di				OR NOT IN_AG.tTCOP_CB_On.GoodQual;
	IN_AG.tTCOP_UPS_CB_On.Di		:= IN_AG.tTCOP_UPS_CB_On.Di			OR NOT IN_AG.tTCOP_UPS_CB_On.GoodQual;
	IN_AG.tECWP_CB_On.Di			:= IN_AG.tECWP_CB_On.Di				OR NOT IN_AG.tECWP_CB_On.GoodQual;
	IN_AG.tECWP_PreH_CB_On.Di		:= IN_AG.tECWP_PreH_CB_On.Di		OR NOT IN_AG.tECWP_PreH_CB_On.GoodQual;
	IN_AG.tChUnit1_CB_On.Di			:= IN_AG.tChUnit1_CB_On.Di			OR NOT IN_AG.tChUnit1_CB_On.GoodQual;
	IN_AG.tChUnit2_CB_On.Di			:= IN_AG.tChUnit2_CB_On.Di			OR NOT IN_AG.tChUnit2_CB_On.GoodQual;
	IN_AG.tChUnit3_CB_On.Di			:= IN_AG.tChUnit3_CB_On.Di			OR NOT IN_AG.tChUnit3_CB_On.GoodQual;
	IN_AG.tChUnit4_CB_On.Di			:= IN_AG.tChUnit4_CB_On.Di			OR NOT IN_AG.tChUnit4_CB_On.GoodQual;
	IN_AG.tPS_EI_CB_On.Di			:= IN_AG.tPS_EI_CB_On.Di			OR NOT IN_AG.tPS_EI_CB_On.GoodQual;
	IN_AG.tSTT_CB_On.Di				:= IN_AG.tSTT_CB_On.Di				OR NOT IN_AG.tSTT_CB_On.GoodQual;
	IN_AG.tENGIA_CB_On.Di			:= IN_AG.tENGIA_CB_On.Di			OR NOT IN_AG.tENGIA_CB_On.GoodQual;
	IN_AG.tECWP_Service_CB_On.Di	:= IN_AG.tECWP_Service_CB_On.Di		OR NOT IN_AG.tECWP_Service_CB_On.GoodQual;
	IN_AG.tPS400V_ENGIA_CB_On.Di	:= IN_AG.tPS400V_ENGIA_CB_On.Di		OR NOT IN_AG.tPS400V_ENGIA_CB_On.GoodQual;
	IN_AG.tUPS_CB_On.Di				:= IN_AG.tUPS_CB_On.Di				OR NOT IN_AG.tUPS_CB_On.GoodQual;
	IN_AG.tENGIA_UPS_CB_On.Di		:= IN_AG.tENGIA_UPS_CB_On.Di		OR NOT IN_AG.tENGIA_UPS_CB_On.GoodQual;
	IN_AG.tCV_Eng_Low.Di			:= IN_AG.tCV_Eng_Low.Di				OR NOT IN_AG.tCV_Eng_Low.GoodQual;
	IN_AG.tCV_TCA_Low.Di			:= IN_AG.tCV_TCA_Low.Di				OR NOT IN_AG.tCV_TCA_Low.GoodQual;
	IN_AG.tCV_MCP_Low.Di			:= IN_AG.tCV_MCP_Low.Di				OR NOT IN_AG.tCV_MCP_Low.GoodQual;

	IN_AG.tBbBlower_FC_Rdy.Di		:= IN_AG.tBbBlower_FC_Rdy.Di		OR NOT IN_AG.tBbBlower_FC_Rdy.GoodQual;

	IN_AG.tAuxV_ModIf_ok.Di			:= IN_AG.tAuxV_ModIf_ok.Di			OR NOT IN_AG.tAuxV_ModIf_ok.GoodQual;
	IN_AG.tAuxV_Aux_ok.Di			:= IN_AG.tAuxV_Aux_ok.Di			OR NOT IN_AG.tAuxV_Aux_ok.GoodQual;
	IN_AG.tL_DayOilSump_Hi.Di		:= IN_AG.tL_DayOilSump_Hi.Di		OR NOT IN_AG.tL_DayOilSump_Hi.GoodQual;
	IN_AG.tDayOilTank_Leck.Di		:= IN_AG.tDayOilTank_Leck.Di		OR NOT IN_AG.tDayOilTank_Leck.GoodQual;
	IN_AG.tL_DayOilTank_Hi.Di		:= IN_AG.tL_DayOilTank_Hi.Di		OR NOT IN_AG.tL_DayOilTank_Hi.GoodQual;

	IN_AG.tL_FreshOilTank_Hi.Di		:= IN_AG.tL_FreshOilTank_Hi.Di		OR NOT IN_AG.tL_FreshOilTank_Hi.GoodQual;
	IN_AG.tOF_FreshOilTank.Di		:= IN_AG.tOF_FreshOilTank.Di		OR NOT IN_AG.tOF_FreshOilTank.GoodQual;
	IN_AG.tLeak_FreshOilPump.Di		:= IN_AG.tLeak_FreshOilPump.Di		OR NOT IN_AG.tLeak_FreshOilPump.GoodQual;
	IN_AG.tLeak_FreshOilTank.Di		:= IN_AG.tLeak_FreshOilTank.Di		OR NOT IN_AG.tLeak_FreshOilTank.GoodQual;
	IN_AG.tOF_WasteOilTank.Di		:= IN_AG.tOF_WasteOilTank.Di		OR NOT IN_AG.tOF_WasteOilTank.GoodQual;
	IN_AG.tLeak_WasteOilPump.Di		:= IN_AG.tLeak_WasteOilPump.Di		OR NOT IN_AG.tLeak_WasteOilPump.GoodQual;
	IN_AG.tLeak_WasteOilTank.Di		:= IN_AG.tLeak_WasteOilTank.Di		OR NOT IN_AG.tLeak_WasteOilTank.GoodQual;
	IN_AG.tGF_OilSystem.Di			:= IN_AG.tGF_OilSystem.Di			OR NOT IN_AG.tGF_OilSystem.GoodQual;

	IN_AG.tCV_GENI_Ok.Di			:= IN_AG.tCV_GENI_Ok.Di				OR NOT IN_AG.tCV_GENI_Ok.GoodQual;
	IN_AG.tCV_ENGIB_Ok.Di			:= IN_AG.tCV_ENGIB_Ok.Di			OR NOT IN_AG.tCV_ENGIB_Ok.GoodQual;
	IN_AG.tCV_TCMI_Ok.Di			:= IN_AG.tCV_TCMI_Ok.Di				OR NOT IN_AG.tCV_TCMI_Ok.GoodQual;
	IN_AG.tCV_TCUS_Ok.Di			:= IN_AG.tCV_TCUS_Ok.Di				OR NOT IN_AG.tCV_TCUS_Ok.GoodQual;
	IN_AG.tCV_JWMI_Ok.Di			:= IN_AG.tCV_JWMI_Ok.Di				OR NOT IN_AG.tCV_JWMI_Ok.GoodQual;
	IN_AG.tCV_OILMI_Ok.Di			:= IN_AG.tCV_OILMI_Ok.Di			OR NOT IN_AG.tCV_OILMI_Ok.GoodQual;
	IN_AG.tCV_M_Ok.Di				:= IN_AG.tCV_M_Ok.Di				OR NOT IN_AG.tCV_M_Ok.GoodQual;
	IN_AG.tCV_A_Ok.Di				:= IN_AG.tCV_A_Ok.Di				OR NOT IN_AG.tCV_A_Ok.GoodQual;
	IN_AG.tCV_AUX_Ok[1].Di			:= IN_AG.tCV_AUX_Ok[1].Di			OR NOT IN_AG.tCV_AUX_Ok[1].GoodQual;
	IN_AG.tCV_AUX_Ok[2].Di			:= IN_AG.tCV_AUX_Ok[2].Di			OR NOT IN_AG.tCV_AUX_Ok[2].GoodQual;
	IN_AG.tCV_AUX_Ok[3].Di			:= IN_AG.tCV_AUX_Ok[3].Di			OR NOT IN_AG.tCV_AUX_Ok[3].GoodQual;
	IN_AG.tCV_AUX_Ok[4].Di			:= IN_AG.tCV_AUX_Ok[4].Di			OR NOT IN_AG.tCV_AUX_Ok[4].GoodQual;
	IN_AG.tCV_AUX_Ok[5].Di			:= IN_AG.tCV_AUX_Ok[5].Di			OR NOT IN_AG.tCV_AUX_Ok[5].GoodQual;

	IN_AG.tOFUP_Centrifuge_CB.Di	:= IN_AG.tOFUP_Centrifuge_CB.Di		OR NOT IN_AG.tOFUP_Centrifuge_CB.GoodQual;
	IN_AG.tOFUP_Filter_CB.Di		:= IN_AG.tOFUP_Filter_CB.Di			OR NOT IN_AG.tOFUP_Filter_CB.GoodQual;

	IN_AG.tBoilerFailure.Di			:= IN_AG.tBoilerFailure.Di			OR NOT IN_AG.tBoilerFailure.GoodQual;
	IN_AG.tSeismicAlarm.Di			:= IN_AG.tSeismicAlarm.Di			OR NOT IN_AG.tSeismicAlarm.GoodQual;

	(* redundant pump options *)
	IF NOT Para.bRedHWP_Active THEN		IN_AG.tHWP_Op.Di	:=	IN_AG.tHWP_Op.Di	OR	NOT IN_AG.tHWP_Op.GoodQual;
	ELSE								IN_AG.tHWP_Op.Di	:=	IN_AG.tHWP1_Op.Di	OR		IN_AG.tHWP2_Op.Di;
	END_IF;

	IF NOT Para.bRedCCWP_Active THEN	IN_AG.tCCWP_Op.Di	:=	IN_AG.tCCWP_Op.Di	OR	NOT IN_AG.tCCWP_Op.GoodQual;
	ELSE								IN_AG.tCCWP_Op.Di	:=	IN_AG.tCCWP1_Op.Di	OR		IN_AG.tCCWP2_Op.Di;
	END_IF;

	IF NOT Para.bRedCC2WP_Active THEN	IN_AG.tCC2WP_Op.Di	:=	IN_AG.tCC2WP_Op.Di	OR	NOT IN_AG.tCC2WP_Op.GoodQual;
	ELSE								IN_AG.tCC2WP_Op.Di	:=	IN_AG.tCC2WP1_Op.Di	OR		IN_AG.tCC2WP2_Op.Di;
	END_IF;

	IF NOT Para.bRedEmCWP_Active THEN	IN_AG.tEmCWP_Op.Di	:=	IN_AG.tEmCWP_Op.Di	OR	NOT IN_AG.tEmCWP_Op.GoodQual;
	ELSE								IN_AG.tEmCWP_Op.Di	:=	IN_AG.tEmCWP1_Op.Di	OR		IN_AG.tEmCWP2_Op.Di;
	END_IF;

	IF NOT IN_AG.tOutAirER_LouClosed.GoodQual THEN
		IN_AG.tOutAirER_LouClosed.Di  :=	TRUE;
	END_IF;
	IF NOT IN_AG.tInAirER_Lou1Closed.GoodQual THEN
		IN_AG.tInAirER_Lou1Closed.Di  :=	TRUE;
	END_IF;
	IF NOT IN_AG.tInAirER_Lou2Closed.GoodQual THEN
		IN_AG.tInAirER_Lou2Closed.Di  :=	TRUE;
	END_IF;

	IN_AG.tFireProtFlap1_InlAir_Opened.Di  := IN_AG.tFireProtFlap1_InlAir_Opened.Di  OR NOT IN_AG.tFireProtFlap1_InlAir_Opened.GoodQual;
	IN_AG.tFireProtFlap2_InlAir_Opened.Di  := IN_AG.tFireProtFlap2_InlAir_Opened.Di  OR NOT IN_AG.tFireProtFlap2_InlAir_Opened.GoodQual;
	IN_AG.tFireProtFlap1_OutlAir_Opened.Di := IN_AG.tFireProtFlap1_OutlAir_Opened.Di OR NOT IN_AG.tFireProtFlap1_OutlAir_Opened.GoodQual;
	IN_AG.tFireProtFlap2_OutlAir_Opened.Di := IN_AG.tFireProtFlap2_OutlAir_Opened.Di OR NOT IN_AG.tFireProtFlap2_OutlAir_Opened.GoodQual;
	IN_AG.tFireProtFlap1_InlAir_Closed.Di  := IN_AG.tFireProtFlap1_InlAir_Closed.Di  OR NOT IN_AG.tFireProtFlap1_InlAir_Closed.GoodQual;
	IN_AG.tFireProtFlap2_InlAir_Closed.Di  := IN_AG.tFireProtFlap2_InlAir_Closed.Di  OR NOT IN_AG.tFireProtFlap2_InlAir_Closed.GoodQual;
	IN_AG.tFireProtFlap1_OutlAir_Closed.Di := IN_AG.tFireProtFlap1_OutlAir_Closed.Di OR NOT IN_AG.tFireProtFlap1_OutlAir_Closed.GoodQual;
	IN_AG.tFireProtFlap2_OutlAir_Closed.Di := IN_AG.tFireProtFlap2_OutlAir_Closed.Di OR NOT IN_AG.tFireProtFlap2_OutlAir_Closed.GoodQual;

	IN_AG.tMCP_AuxPS_CB_Trip.Di		:= IN_AG.tMCP_AuxPS_CB_Trip.Di		OR NOT IN_AG.tMCP_AuxPS_CB_Trip.GoodQual;
	IN_AG.tMCP_AuxPS_CB_On.Di		:= IN_AG.tMCP_AuxPS_CB_On.Di		OR NOT IN_AG.tMCP_AuxPS_CB_On.GoodQual;
	IN_AG.tMCP_AuxPS_GndFault.Di	:= IN_AG.tMCP_AuxPS_GndFault.Di		OR NOT IN_AG.tMCP_AuxPS_GndFault.GoodQual;
	IN_AG.tMCP_FC_GndFault.Di		:= IN_AG.tMCP_FC_GndFault.Di		OR NOT IN_AG.tMCP_FC_GndFault.GoodQual;
	IN_AG.tMIP_FC_GndFault.Di		:= IN_AG.tMIP_FC_GndFault.Di		OR NOT IN_AG.tMIP_FC_GndFault.GoodQual;
	IN_AG.tAuxCP_FC_GndFault.Di		:= IN_AG.tAuxCP_FC_GndFault.Di		OR NOT IN_AG.tAuxCP_FC_GndFault.GoodQual;
	IN_AG.tAuxCP_AuxPS_GndFault.Di	:= IN_AG.tAuxCP_AuxPS_GndFault.Di	OR NOT IN_AG.tAuxCP_AuxPS_GndFault.GoodQual;
	IN_AG.tAuxCP_AuxPS_CB_Trip.Di	:= IN_AG.tAuxCP_AuxPS_CB_Trip.Di	OR NOT IN_AG.tAuxCP_AuxPS_CB_Trip.GoodQual;
	IN_AG.tAuxCP_AuxPS_CB_On.Di		:= IN_AG.tAuxCP_AuxPS_CB_On.Di		OR NOT IN_AG.tAuxCP_AuxPS_CB_On.GoodQual;

	IN_AG.tBatChargeDev_Ok.Di		:= IN_AG.tBatChargeDev_Ok.Di		OR NOT IN_AG.tBatChargeDev_Ok.GoodQual;
	FOR iIdx_CtrlBat := 1 TO iNum_CtrlBatMon DO
		IN_AG.tCtrlBat_ChargeDev_Ok[iIdx_CtrlBat].Di	:=	IN_AG.tCtrlBat_ChargeDev_Ok[iIdx_CtrlBat].Di	OR NOT IN_AG.tCtrlBat_ChargeDev_Ok[iIdx_CtrlBat].GoodQual;
	END_FOR;

	IN_AG.tLeak_OilExtensionTank1.Di	:= IN_AG.tLeak_OilExtensionTank1.Di	OR NOT IN_AG.tLeak_OilExtensionTank1.GoodQual;
	IN_AG.tLeak_OilExtensionTank2.Di	:= IN_AG.tLeak_OilExtensionTank2.Di	OR NOT IN_AG.tLeak_OilExtensionTank2.GoodQual;
	IN_AG.tLeak_OilExtensionTank3.Di	:= IN_AG.tLeak_OilExtensionTank3.Di	OR NOT IN_AG.tLeak_OilExtensionTank3.GoodQual;

//	IN_AG.x.Di		:=	IN_AG.x.Di		OR	NOT IN_AG.x.GoodQual;

END_PROGRAM
```

#### default_AG.var
```iecst
VAR
	iIdx_CtrlBat : USINT;
END_VAR
```

### Program Logical/AuxiliariesGeneral/default_AG_TC2 (IEC, version 4.03.0) - default_TC2

#### default_AG_TC2Cyclic.st
```iecst
(*******************************************************************************
default		value set

This code is confidential AND proprietary to the INNIO Company.
It may NOT be used in any form, or reproduced in any manner,
without the express written permission of the INNIO Company.
Copyright, INNIO Company, 2019

Customized modifications: -
------------------------

History:
-------
V4.03.0 03.11.2015	lettenb.	new für TC2

Instructions FOR use:
--------------------
Outstandings:
------------
*******************************************************************************)
PROGRAM _CYCLIC

	(* default TRUE setting for not existing Di's *)
	IN_AG.tEO_Level_Lo_TC2.Di		:=	IN_AG.tEO_Level_Lo_TC2.Di		OR	NOT IN_AG.tEO_Level_Lo_TC2.GoodQual;

	//	IN_AG.x.Di		:=	IN_AG.x.Di		OR	NOT IN_AG.x.GoodQual;

END_PROGRAM
```

### Program Logical/AuxiliariesGeneral/AuxGnl (IEC, version 4.25.0) - auxiliaries general
